// Mitsubishi GX Works2 project: e01   PLC: Q02/Q02H

PROGRAM MAIN
VAR
  자기_1 : 자기;
  디카운터_1 : 디카운터;
END_VAR
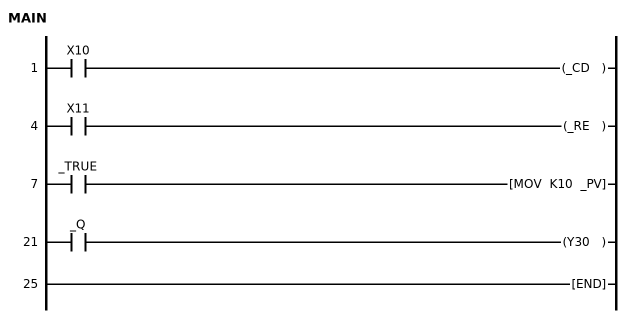
; FB BLK START 디카운터(디카운터_1)
1     LD      X10
      OUT     _CD
4     LD      X11
      OUT     _RE
7     LD      _TRUE
      MOV     K10 _PV
; FB START
; FB_NAME 디카운터
; INSTANCE_NAME 디카운터_1
; FB IN_B:CD
; FB OUT_Q:B
; FB IN_B:RE
; FB OUT_CV:W
; FB IN_W:PV
; FB END
21    LD      _Q
      OUT     Y30
; FB BLK END
25    END
END_PROGRAM

FUNCTION_BLOCK 자기
VAR_INPUT
  SSP : BOOL;
  SST : BOOL;
END_VAR
VAR_OUTPUT
  OOUT : BOOL;
END_VAR
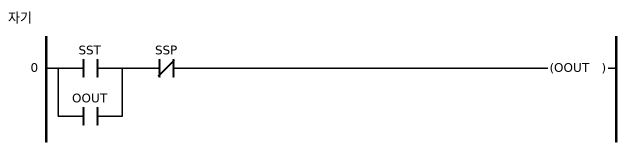
0     LD      SST
      OR      OOUT
      ANI     SSP
      OUT     OOUT
END_FUNCTION_BLOCK

FUNCTION_BLOCK 디카운터
VAR_INPUT
  CD : BOOL;
  RE : BOOL;
  PV : INT;
END_VAR
VAR_OUTPUT
  Q : BOOL;
  CV : INT;
END_VAR
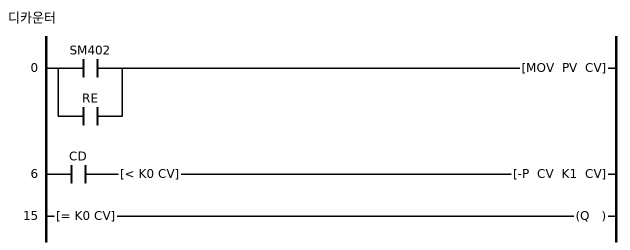
0     LD      SM402
      OR      RE
      MOV     PV CV
6     LD      CD
      AND<    K0 CV
      -P      CV K1 CV
15    LD=     K0 CV
      OUT     Q
END_FUNCTION_BLOCK
